{attribute addProperty BoxType "EL6021-0000-0018"}
{attribute addProperty Id "COM_TxPDO_Map_InputsAT %I*COM_TxPDO_Map_Inputs_85D1D733192240COM_RxPDO_Map_OutputsAT %Q*COM_RxPDO_Map_Outputs_AC29F8FC192240WcStateAT %I*WcState_F855686C1620InfoDataAT %I*InfoData_BC63D37F80100"}
{attribute addProperty CRC "4202498057"}
{attribute addProperty SizeInBites "480"}
{attribute addProperty SizeInBytes "60"}
TYPE EL6021_2B16659A :
STRUCT
	{attribute addProperty Name "COM_TxPDO_Map_Inputs"}
	COM_TxPDO_Map_Inputs : COM_TxPDO_Map_Inputs_85D1D733;
	{attribute addProperty Name "COM_RxPDO_Map_Outputs"}
	COM_RxPDO_Map_Outputs : COM_RxPDO_Map_Outputs_AC29F8FC;
	{attribute addProperty Name "WcState"}
	WcState : WcState_F855686C;
	{attribute addProperty Name "InfoData"}
	InfoData : InfoData_BC63D37F;
END_STRUCT
END_TYPE

(* stored: Version 1.2.0.0, ProductVersion 3.1.4024.9
   DUT EL6021_2B16659A: Id {e07839f3-3a69-46b4-904f-68d85487e61c} *)
